PROGRAM P_Demo_F_BA_RVal
VAR
    argFValue                      : REAL                           := 0.0; // fValue
    fnReturn                       : U_BA_ClassValue; // 返回值
END_VAR

// =============================================================================
// Tc3_BA2_Common.F_BA_RVal 演示程序
// =============================================================================
// 场景：温度 / 压力 / 流量等 REAL 测点统一封装为带单位（℃ / kPa / m³/h）的 ClassValue 上报。
//
// 价值：一次性把"数值 + 单位 + 状态"组合进同一结构，简化下游解析。
//
// 验证：登录 PLC 后，按例程内变量在线写值；监视输出 / 返回值，结合 §1 功能
//       简述的预期行为对照（详见配套 .md 文档 §7 业务场景）。
//
// 验证步骤：
//   1. 右键 PLC 项目下 POUs 文件夹 → Add → Existing Item → 选本 .TcPOU 文件
//   2. 引用 Tc3_BA2_Common（References → Add library）
//   3. 编译 → 登录 → 运行；按上方『验证』指引在线写值观察
// =============================================================================

fnReturn := F_BA_RVal(
    fValue                   := argFValue
);

END_PROGRAM

(* stored: Version 1.1.0.1, ProductVersion 3.1.4024.5
   POU P_Demo_F_BA_RVal: Id {908970c3-74a6-5944-966c-0e41a4ad2429}, SpecialFunc None *)
